FUNCTION_BLOCK fb_Slitter EXTENDS FB_Generic
VAR_INPUT
END_VAR
VAR_OUTPUT
END_VAR
VAR
	iManSlitStep	:INT;
	rtPedalSlite	:R_TRIG;
	tonPedalSlite	:TON;
	bTmp1: BOOL;
	bManSlitRunning: BOOL;
	i: INT;
	fbSlitterAct	:FB_SlitterAct;
END_VAR

SUPER^();
//tonPedalSlite(IN:=In_pedal1_Slitter , PT:=T#2S , Q=> , ET=> );

stFolder.Status.Slitter_AtHome	:=In_sigSlitLmt0;

fbSlitterAct(Done=> );

Out_SlitterFwd	:=fbSlitterAct.bOutSlitterFwd AND In_sigBtmApron_SlideFWD AND In_sigBtmApron_FoldHome;
Out_SlitterBwd	:=fbSlitterAct.bOutSlitterBwd AND In_sigBtmApron_SlideFWD AND In_sigBtmApron_FoldHome;



IF NOT stFolder.Status.SlitterAtSlow AND NOT Hmi_bArray[88] AND NOT Hmi_bArray[89] THEN
	Out_SlitterSpeed:= TRUE;
ELSE
	Out_SlitterSpeed:= FALSE;
END_IF		

IF Hmi_bArray[88] THEN 
	Out_SlitterFwd := TRUE;
END_IF

IF Hmi_bArray[89] THEN 
	Out_SlitterBwd := TRUE;
END_IF

ACTION A_AutoRun:

END_ACTION

ACTION A_ManualRun:

END_ACTION

{attribute 'object_name' := 'M_Execute'}
METHOD M_Execute

VAR
	
END_VAR
CASE fbUnitModeManager.eModeStatus OF
	ePMLProtUnitMode_Production:		//Production
		;
		
	ePMLProtUnitMode_Maintenance:		
		//
		;
		ePMLUnitMode_Auto:
		IF stFolderCom.TaskSlitter =eTask_SlitterAct THEN
			IF fbSlitterAct.Done THEN
				stFolderCom.TaskSlitter	:=eTask_NULL;
			END_IF
		END_IF
	ePMLUnitMode_SemiAuto:
		i:=334;
		IF stFolderCom.TaskSlitter =eTask_SlitterAct THEN
			IF fbSlitterAct.Done THEN
				stFolderCom.TaskSlitter	:=eTask_NULL;
			END_IF
		END_IF
	ePMLUnitMode_AutoSlitter:
		i:=339;
		IF stFolderCom.TaskSlitter =eTask_SlitterAct THEN
			IF fbSlitterAct.Done THEN
				stFolderCom.TaskSlitter	:=eTask_NULL;
			END_IF
		END_IF
	ePMLProtUnitMode_Manual:		//Manual
		A_ManualRun();
		stFolderCom.TaskSlitter :=eTask_SlitterAct;


		//Out_SlitterFwd	:=In_pedal1_Slitter AND NOT In_sigSlitSlw1 AND NOT In_sigSlitLmt1 ;
		//Out_SlitterBwd	:=In_pedal1_SlitterBack;
		
		

		
END_CASE
END_METHOD

END_FUNCTION_BLOCK

(* stored: Version 1.1.0.1, ProductVersion 3.1.4024.15
   POU fb_Slitter: Id {78ce88af-4045-4c39-86ae-b95d1f8aa49b}, SpecialFunc None
   Action A_AutoRun: Id {8b28f82b-5989-4ee0-8606-98f8fb9ce2bb}
   Action A_ManualRun: Id {cfd41d8d-2eb5-4692-9fb9-6bc421709b26}
   Method M_Execute: Id {69ace4f9-def2-4eea-b4be-ca3a25d7688f} *)
